Xinje XCPPro project, PLC1: XC3-60 (software 3.3k)

PROGRAM Ladder

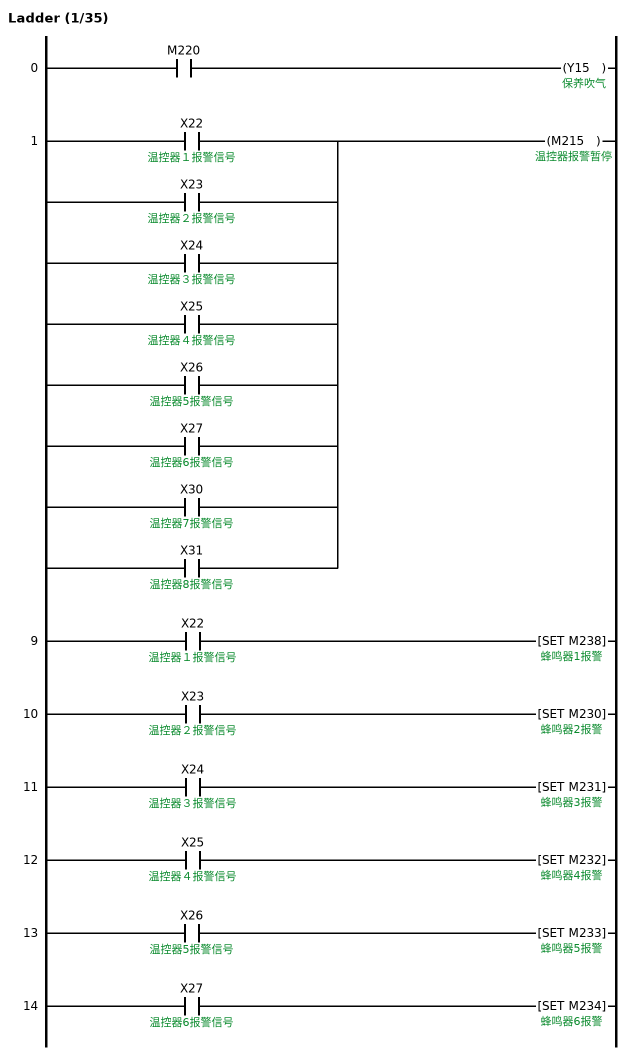
LD     M220
OUT    Y15	; 保养吹气 
LD     X22	; 温控器１报警信号
OR     X23	; 温控器２报警信号
OR     X24	; 温控器３报警信号
OR     X25	; 温控器４报警信号
OR     X26	; 温控器5报警信号
OR     X27	; 温控器6报警信号
OR     X30	; 温控器7报警信号
OR     X31	; 温控器8报警信号
OUT    M215	; 温控器报警暂停
LD     X22	; 温控器１报警信号
SET    M238	; 蜂鸣器1报警
LD     X23	; 温控器２报警信号
SET    M230	; 蜂鸣器2报警
LD     X24	; 温控器３报警信号
SET    M231	; 蜂鸣器3报警
LD     X25	; 温控器４报警信号
SET    M232	; 蜂鸣器4报警
LD     X26	; 温控器5报警信号
SET    M233	; 蜂鸣器5报警
LD     X27	; 温控器6报警信号
SET    M234	; 蜂鸣器6报警

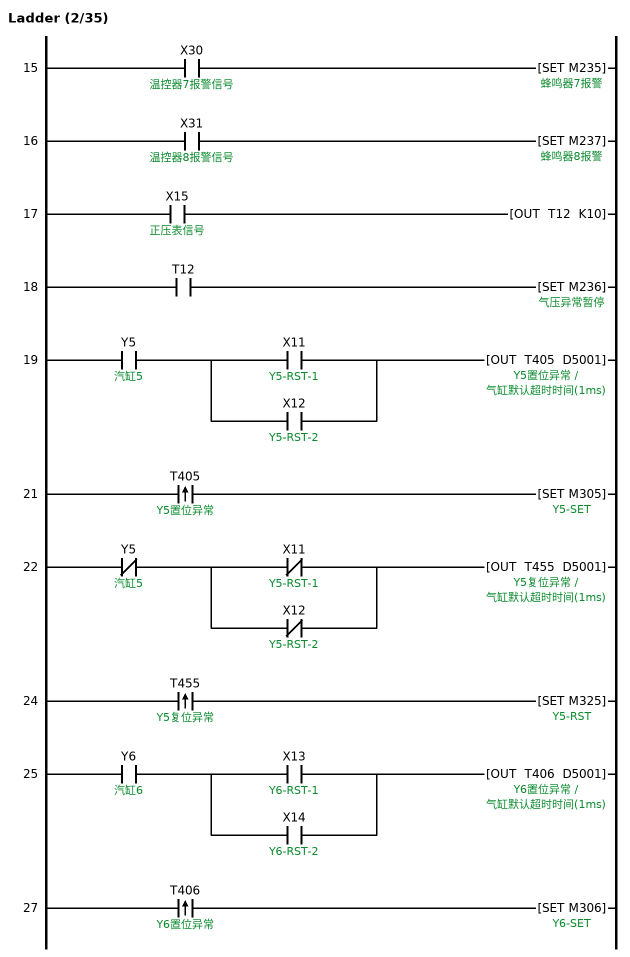
LD     X30	; 温控器7报警信号
SET    M235	; 蜂鸣器7报警
LD     X31	; 温控器8报警信号
SET    M237	; 蜂鸣器8报警
LD     X15	; 正压表信号
OUT    T12 K10
LD     T12
SET    M236	; 气压异常暂停
LD     Y5	; 汽缸5
LD     X11	; Y5-RST-1
OR     X12	; Y5-RST-2
ANB
OUT    T405 D5001	; Y5置位异常 / 气缸默认超时时间(1ms)
LDP    T405	; Y5置位异常
SET    M305	; Y5-SET
LDI    Y5	; 汽缸5
LDI    X11	; Y5-RST-1
ORI    X12	; Y5-RST-2
ANB
OUT    T455 D5001	; Y5复位异常 / 气缸默认超时时间(1ms)
LDP    T455	; Y5复位异常
SET    M325	; Y5-RST
LD     Y6	; 汽缸6
LD     X13	; Y6-RST-1
OR     X14	; Y6-RST-2
ANB
OUT    T406 D5001	; Y6置位异常 / 气缸默认超时时间(1ms)
LDP    T406	; Y6置位异常
SET    M306	; Y6-SET

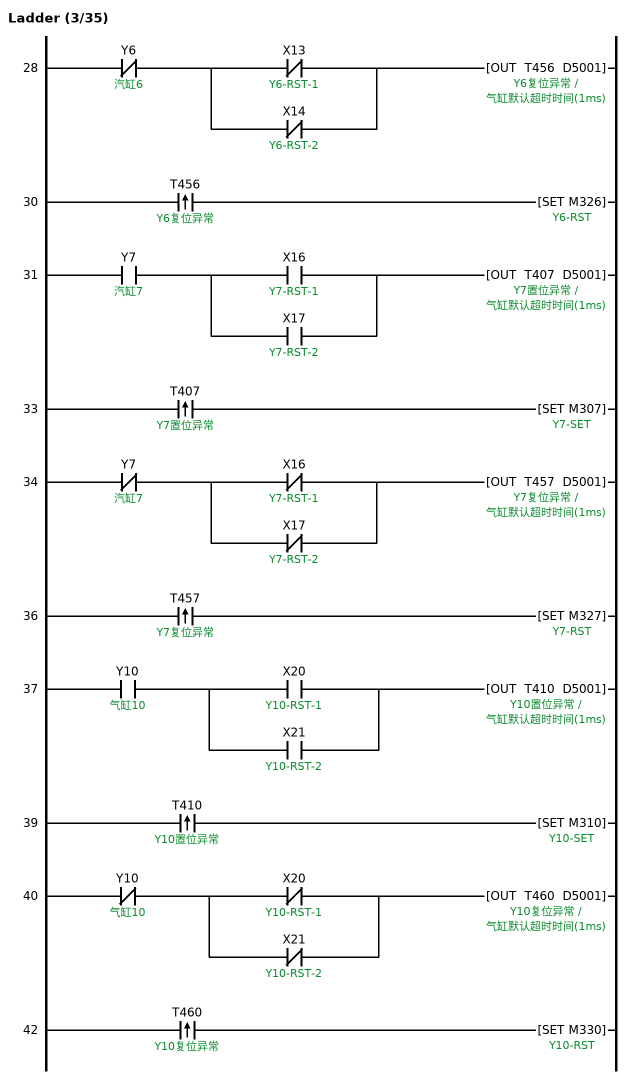
LDI    Y6	; 汽缸6
LDI    X13	; Y6-RST-1
ORI    X14	; Y6-RST-2
ANB
OUT    T456 D5001	; Y6复位异常 / 气缸默认超时时间(1ms)
LDP    T456	; Y6复位异常
SET    M326	; Y6-RST
LD     Y7	; 汽缸7
LD     X16	; Y7-RST-1
OR     X17	; Y7-RST-2
ANB
OUT    T407 D5001	; Y7置位异常 / 气缸默认超时时间(1ms)
LDP    T407	; Y7置位异常
SET    M307	; Y7-SET
LDI    Y7	; 汽缸7
LDI    X16	; Y7-RST-1
ORI    X17	; Y7-RST-2
ANB
OUT    T457 D5001	; Y7复位异常 / 气缸默认超时时间(1ms)
LDP    T457	; Y7复位异常
SET    M327	; Y7-RST
LD     Y10	; 气缸10
LD     X20	; Y10-RST-1
OR     X21	; Y10-RST-2
ANB
OUT    T410 D5001	; Y10置位异常 / 气缸默认超时时间(1ms)
LDP    T410	; Y10置位异常
SET    M310	; Y10-SET
LDI    Y10	; 气缸10
LDI    X20	; Y10-RST-1
ORI    X21	; Y10-RST-2
ANB
OUT    T460 D5001	; Y10复位异常 / 气缸默认超时时间(1ms)
LDP    T460	; Y10复位异常
SET    M330	; Y10-RST

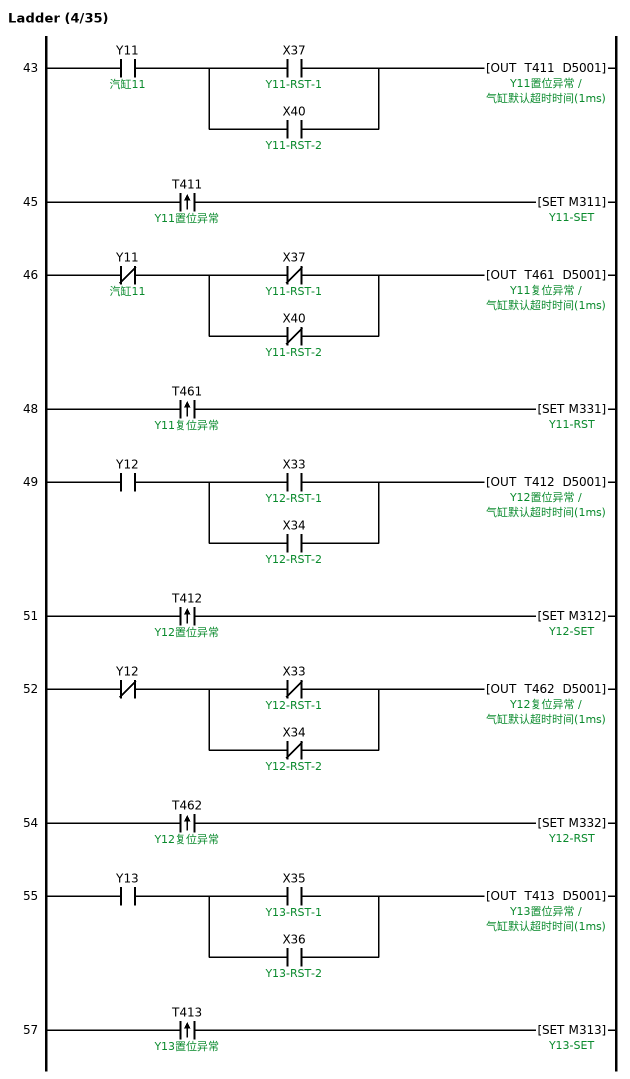
LD     Y11	; 汽缸11
LD     X37	; Y11-RST-1
OR     X40	; Y11-RST-2
ANB
OUT    T411 D5001	; Y11置位异常 / 气缸默认超时时间(1ms)
LDP    T411	; Y11置位异常
SET    M311	; Y11-SET
LDI    Y11	; 汽缸11
LDI    X37	; Y11-RST-1
ORI    X40	; Y11-RST-2
ANB
OUT    T461 D5001	; Y11复位异常 / 气缸默认超时时间(1ms)
LDP    T461	; Y11复位异常
SET    M331	; Y11-RST
LD     Y12
LD     X33	; Y12-RST-1
OR     X34	; Y12-RST-2
ANB
OUT    T412 D5001	; Y12置位异常 / 气缸默认超时时间(1ms)
LDP    T412	; Y12置位异常
SET    M312	; Y12-SET
LDI    Y12
LDI    X33	; Y12-RST-1
ORI    X34	; Y12-RST-2
ANB
OUT    T462 D5001	; Y12复位异常 / 气缸默认超时时间(1ms)
LDP    T462	; Y12复位异常
SET    M332	; Y12-RST
LD     Y13
LD     X35	; Y13-RST-1
OR     X36	; Y13-RST-2
ANB
OUT    T413 D5001	; Y13置位异常 / 气缸默认超时时间(1ms)
LDP    T413	; Y13置位异常
SET    M313	; Y13-SET

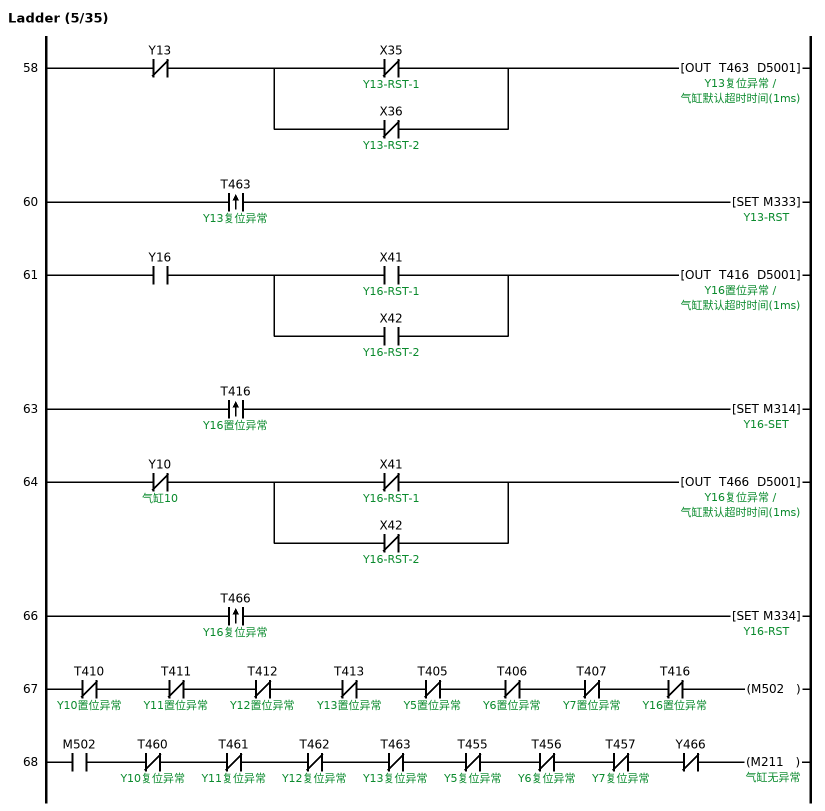
LDI    Y13
LDI    X35	; Y13-RST-1
ORI    X36	; Y13-RST-2
ANB
OUT    T463 D5001	; Y13复位异常 / 气缸默认超时时间(1ms)
LDP    T463	; Y13复位异常
SET    M333	; Y13-RST
LD     Y16
LD     X41	; Y16-RST-1
OR     X42	; Y16-RST-2
ANB
OUT    T416 D5001	; Y16置位异常 / 气缸默认超时时间(1ms)
LDP    T416	; Y16置位异常
SET    M314	; Y16-SET
LDI    Y10	; 气缸10
LDI    X41	; Y16-RST-1
ORI    X42	; Y16-RST-2
ANB
OUT    T466 D5001	; Y16复位异常 / 气缸默认超时时间(1ms)
LDP    T466	; Y16复位异常
SET    M334	; Y16-RST
LDI    T410	; Y10置位异常
ANI    T411	; Y11置位异常
ANI    T412	; Y12置位异常
ANI    T413	; Y13置位异常
ANI    T405	; Y5置位异常
ANI    T406	; Y6置位异常
ANI    T407	; Y7置位异常
ANI    T416	; Y16置位异常
OUT    M502
LD     M502
ANI    T460	; Y10复位异常
ANI    T461	; Y11复位异常
ANI    T462	; Y12复位异常
ANI    T463	; Y13复位异常
ANI    T455	; Y5复位异常
ANI    T456	; Y6复位异常
ANI    T457	; Y7复位异常
ANI    Y466
OUT    M211	; 气缸无异常

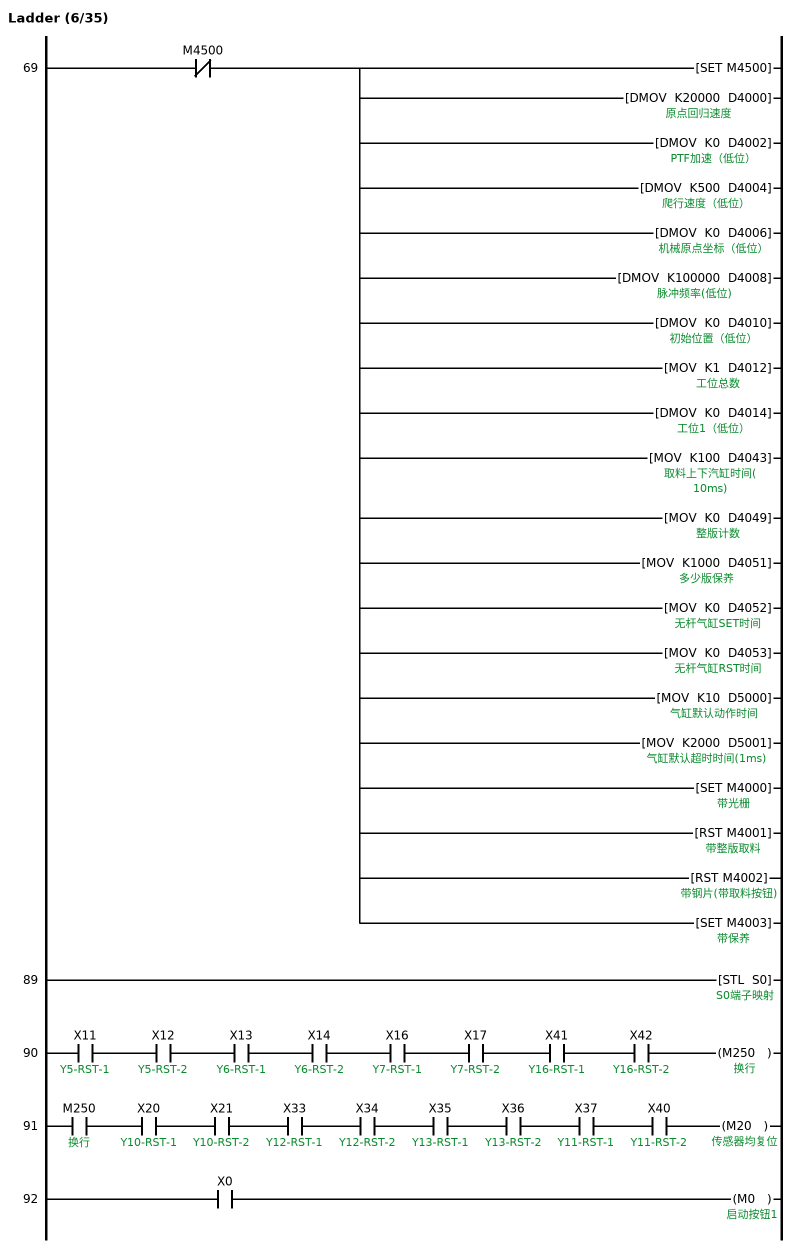
LDI    M4500
SET    M4500
DMOV   K20000 D4000	; 原点回归速度
DMOV   K0 D4002	; PTF加速（低位）
DMOV   K500 D4004	; 爬行速度（低位）
DMOV   K0 D4006	; 机械原点坐标（低位）
DMOV   K100000 D4008	; 脉冲频率(低位)
DMOV   K0 D4010	; 初始位置（低位）
MOV    K1 D4012	; 工位总数
DMOV   K0 D4014	; 工位1（低位）
MOV    K100 D4043	; 取料上下汽缸时间(10ms)
MOV    K0 D4049	; 整版计数
MOV    K1000 D4051	; 多少版保养
MOV    K0 D4052	; 无杆气缸SET时间
MOV    K0 D4053	; 无杆气缸RST时间
MOV    K10 D5000	; 气缸默认动作时间
MOV    K2000 D5001	; 气缸默认超时时间(1ms)
SET    M4000	; 带光栅
RST    M4001	; 带整版取料
RST    M4002	; 带钢片(带取料按钮)
SET    M4003	; 带保养
STL    S0	; S0端子映射
LD     X11	; Y5-RST-1
AND    X12	; Y5-RST-2
AND    X13	; Y6-RST-1
AND    X14	; Y6-RST-2
AND    X16	; Y7-RST-1
AND    X17	; Y7-RST-2
AND    X41	; Y16-RST-1
AND    X42	; Y16-RST-2
OUT    M250	; 换行
LD     M250	; 换行
AND    X20	; Y10-RST-1
AND    X21	; Y10-RST-2
AND    X33	; Y12-RST-1
AND    X34	; Y12-RST-2
AND    X35	; Y13-RST-1
AND    X36	; Y13-RST-2
AND    X37	; Y11-RST-1
AND    X40	; Y11-RST-2
OUT    M20	; 传感器均复位
LD     X0
OUT    M0	; 启动按钮1

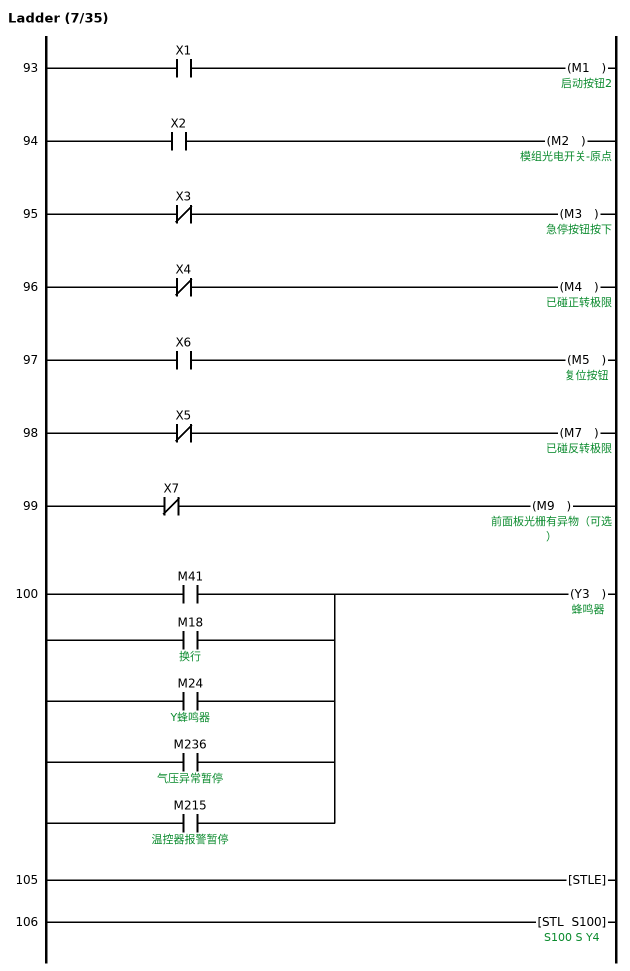
LD     X1
OUT    M1	; 启动按钮2
LD     X2
OUT    M2	; 模组光电开关-原点
LDI    X3
OUT    M3	; 急停按钮按下
LDI    X4
OUT    M4	; 已碰正转极限
LD     X6
OUT    M5	; 复位按钮
LDI    X5
OUT    M7	; 已碰反转极限
LDI    X7
OUT    M9	; 前面板光栅有异物（可选）
LD     M41
OR     M18	; 换行
OR     M24	; Y蜂鸣器
OR     M236	; 气压异常暂停
OR     M215	; 温控器报警暂停
OUT    Y3	; 蜂鸣器
STLE
STL    S100	; S100 S Y4

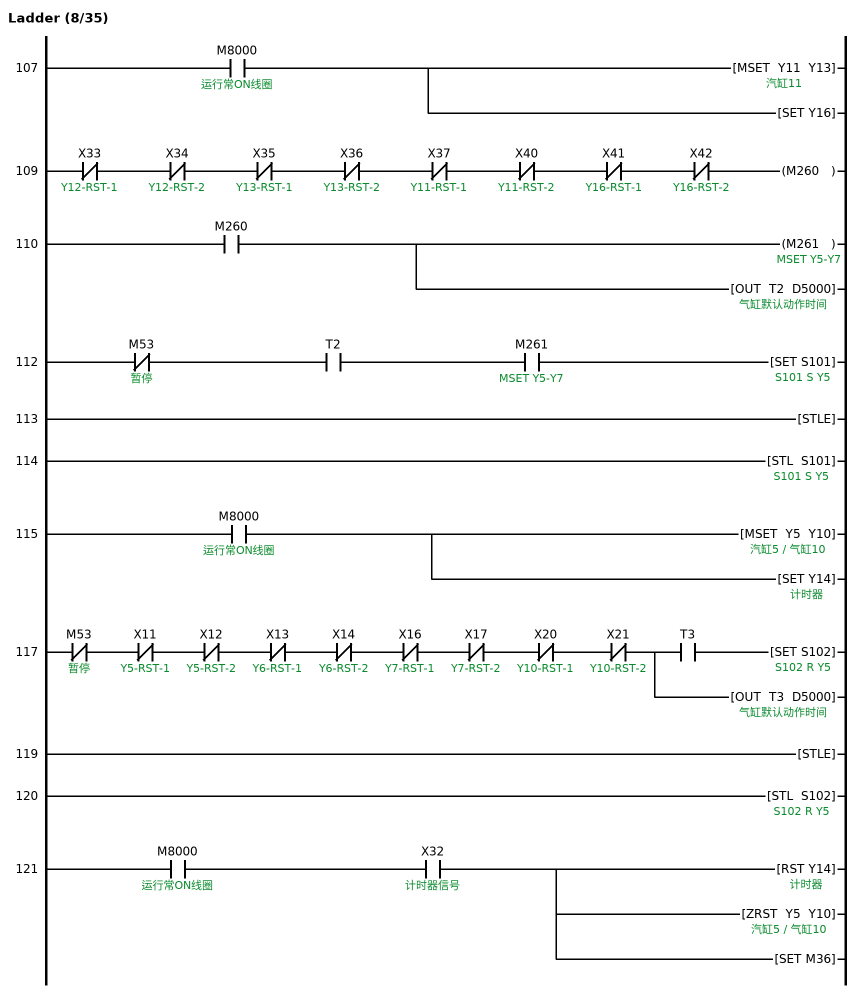
LD     M8000	; 运行常ON线圈
MSET   Y11 Y13	; 汽缸11
SET    Y16
LDI    X33	; Y12-RST-1
ANI    X34	; Y12-RST-2
ANI    X35	; Y13-RST-1
ANI    X36	; Y13-RST-2
ANI    X37	; Y11-RST-1
ANI    X40	; Y11-RST-2
ANI    X41	; Y16-RST-1
ANI    X42	; Y16-RST-2
OUT    M260
LD     M260
OUT    M261	; MSET Y5-Y7
OUT    T2 D5000	; 气缸默认动作时间
LDI    M53	; 暂停
AND    T2
AND    M261	; MSET Y5-Y7
SET    S101	; S101 S Y5
STLE
STL    S101	; S101 S Y5
LD     M8000	; 运行常ON线圈
MSET   Y5 Y10	; 汽缸5 / 气缸10
SET    Y14	; 计时器
LDI    M53	; 暂停
ANI    X11	; Y5-RST-1
ANI    X12	; Y5-RST-2
ANI    X13	; Y6-RST-1
ANI    X14	; Y6-RST-2
ANI    X16	; Y7-RST-1
ANI    X17	; Y7-RST-2
ANI    X20	; Y10-RST-1
ANI    X21	; Y10-RST-2
MPS
AND    T3
SET    S102	; S102 R Y5 
MPP
OUT    T3 D5000	; 气缸默认动作时间
STLE
STL    S102	; S102 R Y5 
LD     M8000	; 运行常ON线圈
AND    X32	; 计时器信号
RST    Y14	; 计时器
ZRST   Y5 Y10	; 汽缸5 / 气缸10
SET    M36

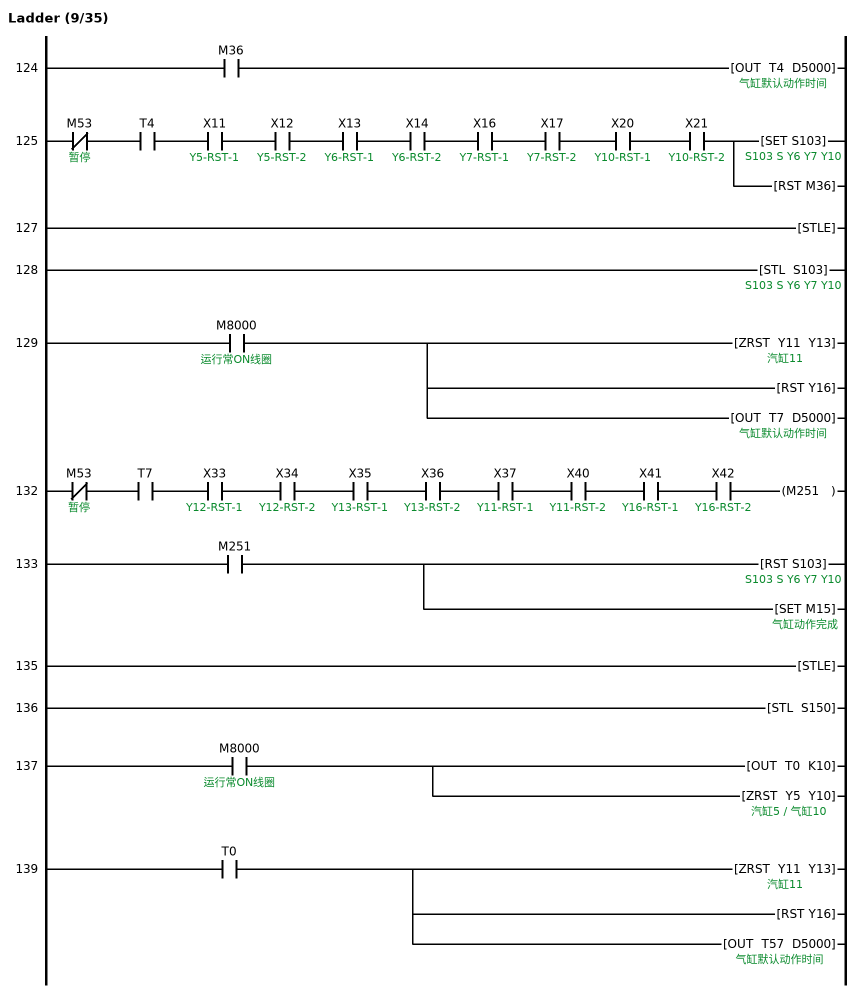
LD     M36
OUT    T4 D5000	; 气缸默认动作时间
LDI    M53	; 暂停
AND    T4
AND    X11	; Y5-RST-1
AND    X12	; Y5-RST-2
AND    X13	; Y6-RST-1
AND    X14	; Y6-RST-2
AND    X16	; Y7-RST-1
AND    X17	; Y7-RST-2
AND    X20	; Y10-RST-1
AND    X21	; Y10-RST-2
SET    S103	; S103 S Y6 Y7 Y10 
RST    M36
STLE
STL    S103	; S103 S Y6 Y7 Y10 
LD     M8000	; 运行常ON线圈
ZRST   Y11 Y13	; 汽缸11
RST    Y16
OUT    T7 D5000	; 气缸默认动作时间
LDI    M53	; 暂停
AND    T7
AND    X33	; Y12-RST-1
AND    X34	; Y12-RST-2
AND    X35	; Y13-RST-1
AND    X36	; Y13-RST-2
AND    X37	; Y11-RST-1
AND    X40	; Y11-RST-2
AND    X41	; Y16-RST-1
AND    X42	; Y16-RST-2
OUT    M251
LD     M251
RST    S103	; S103 S Y6 Y7 Y10 
SET    M15	; 气缸动作完成
STLE
STL    S150
LD     M8000	; 运行常ON线圈
OUT    T0 K10
ZRST   Y5 Y10	; 汽缸5 / 气缸10
LD     T0
ZRST   Y11 Y13	; 汽缸11
RST    Y16
OUT    T57 D5000	; 气缸默认动作时间

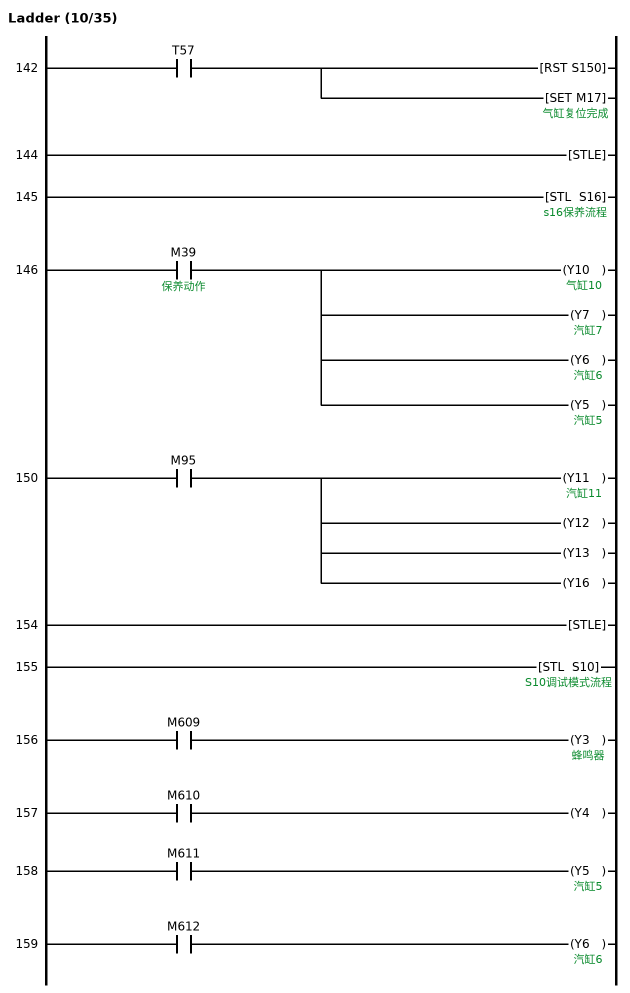
LD     T57
RST    S150
SET    M17	; 气缸复位完成
STLE
STL    S16	; s16保养流程
LD     M39	; 保养动作
OUT    Y10	; 气缸10
OUT    Y7	; 汽缸7
OUT    Y6	; 汽缸6
OUT    Y5	; 汽缸5
LD     M95
OUT    Y11	; 汽缸11
OUT    Y12
OUT    Y13
OUT    Y16
STLE
STL    S10	; S10调试模式流程
LD     M609
OUT    Y3	; 蜂鸣器
LD     M610
OUT    Y4
LD     M611
OUT    Y5	; 汽缸5
LD     M612
OUT    Y6	; 汽缸6

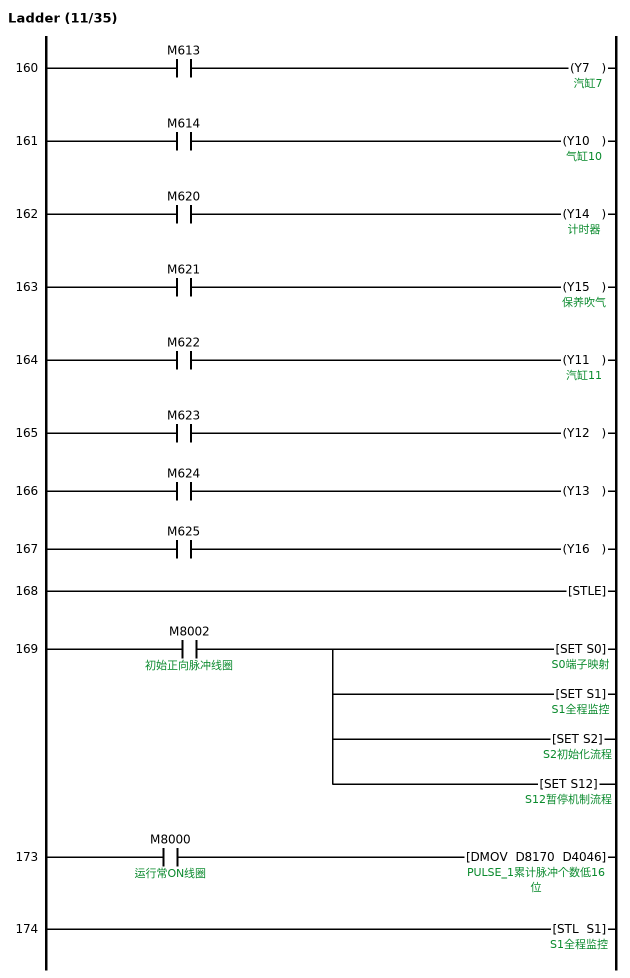
LD     M613
OUT    Y7	; 汽缸7
LD     M614
OUT    Y10	; 气缸10
LD     M620
OUT    Y14	; 计时器
LD     M621
OUT    Y15	; 保养吹气 
LD     M622
OUT    Y11	; 汽缸11
LD     M623
OUT    Y12
LD     M624
OUT    Y13
LD     M625
OUT    Y16
STLE
LD     M8002	; 初始正向脉冲线圈
SET    S0	; S0端子映射
SET    S1	; S1全程监控
SET    S2	; S2初始化流程
SET    S12	; S12暂停机制流程
LD     M8000	; 运行常ON线圈
DMOV   D8170 D4046	; PULSE_1累计脉冲个数低16位
STL    S1	; S1全程监控

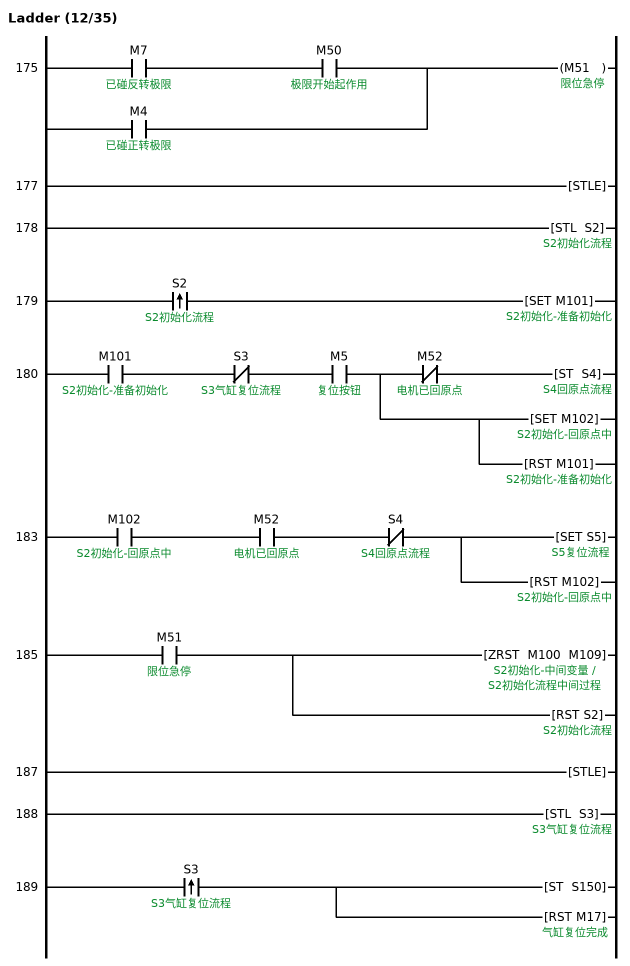
LD     M7	; 已碰反转极限
AND    M50	; 极限开始起作用
OR     M4	; 已碰正转极限
OUT    M51	; 限位急停
STLE
STL    S2	; S2初始化流程
LDP    S2	; S2初始化流程
SET    M101	; S2初始化-准备初始化
LD     M101	; S2初始化-准备初始化
ANI    S3	; S3气缸复位流程
AND    M5	; 复位按钮
MPS
ANI    M52	; 电机已回原点
ST     S4	; S4回原点流程
MPP
SET    M102	; S2初始化-回原点中
RST    M101	; S2初始化-准备初始化
LD     M102	; S2初始化-回原点中
AND    M52	; 电机已回原点
ANI    S4	; S4回原点流程
SET    S5	; S5复位流程
RST    M102	; S2初始化-回原点中
LD     M51	; 限位急停
ZRST   M100 M109	; S2初始化-中间变量 / S2初始化流程中间过程
RST    S2	; S2初始化流程
STLE
STL    S3	; S3气缸复位流程
LDP    S3	; S3气缸复位流程
ST     S150
RST    M17	; 气缸复位完成

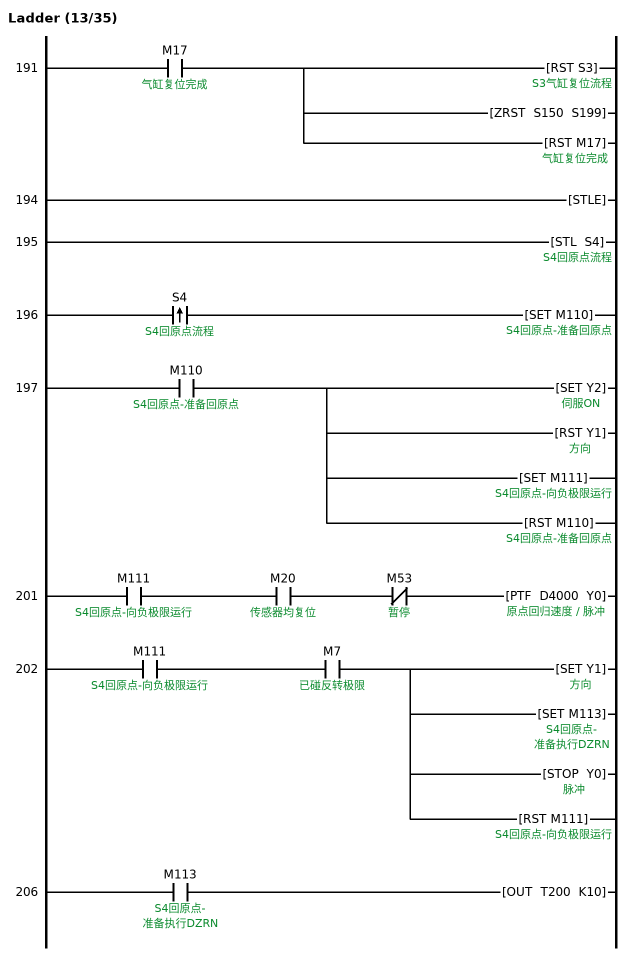
LD     M17	; 气缸复位完成
RST    S3	; S3气缸复位流程
ZRST   S150 S199
RST    M17	; 气缸复位完成
STLE
STL    S4	; S4回原点流程
LDP    S4	; S4回原点流程
SET    M110	; S4回原点-准备回原点
LD     M110	; S4回原点-准备回原点
SET    Y2	; 伺服ON
RST    Y1	; 方向
SET    M111	; S4回原点-向负极限运行
RST    M110	; S4回原点-准备回原点
LD     M111	; S4回原点-向负极限运行
AND    M20	; 传感器均复位
ANI    M53	; 暂停
PTF    D4000 Y0	; 原点回归速度 / 脉冲
LD     M111	; S4回原点-向负极限运行
AND    M7	; 已碰反转极限
SET    Y1	; 方向
SET    M113	; S4回原点-准备执行DZRN
STOP   Y0	; 脉冲
RST    M111	; S4回原点-向负极限运行
LD     M113	; S4回原点-准备执行DZRN
OUT    T200 K10

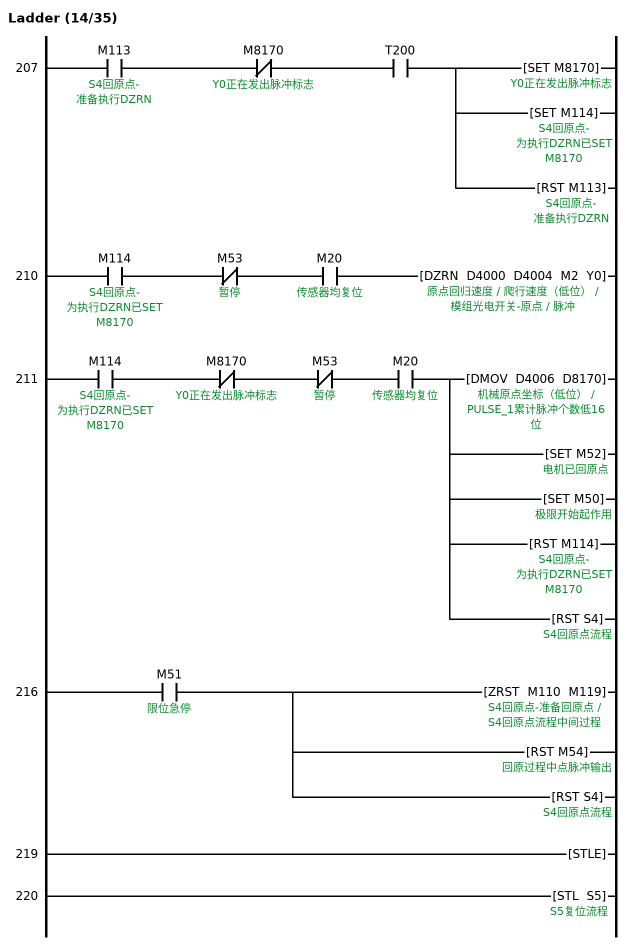
LD     M113	; S4回原点-准备执行DZRN
ANI    M8170	; Y0正在发出脉冲标志
AND    T200
SET    M8170	; Y0正在发出脉冲标志
SET    M114	; S4回原点-为执行DZRN已SET M8170
RST    M113	; S4回原点-准备执行DZRN
LD     M114	; S4回原点-为执行DZRN已SET M8170
ANI    M53	; 暂停
AND    M20	; 传感器均复位
DZRN   D4000 D4004 M2 Y0	; 原点回归速度 / 爬行速度（低位） / 模组光电开关-原点 / 脉冲
LD     M114	; S4回原点-为执行DZRN已SET M8170
ANI    M8170	; Y0正在发出脉冲标志
ANI    M53	; 暂停
AND    M20	; 传感器均复位
DMOV   D4006 D8170	; 机械原点坐标（低位） / PULSE_1累计脉冲个数低16位
SET    M52	; 电机已回原点
SET    M50	; 极限开始起作用
RST    M114	; S4回原点-为执行DZRN已SET M8170
RST    S4	; S4回原点流程
LD     M51	; 限位急停
ZRST   M110 M119	; S4回原点-准备回原点 / S4回原点流程中间过程
RST    M54	; 回原过程中点脉冲输出
RST    S4	; S4回原点流程
STLE
STL    S5	; S5复位流程

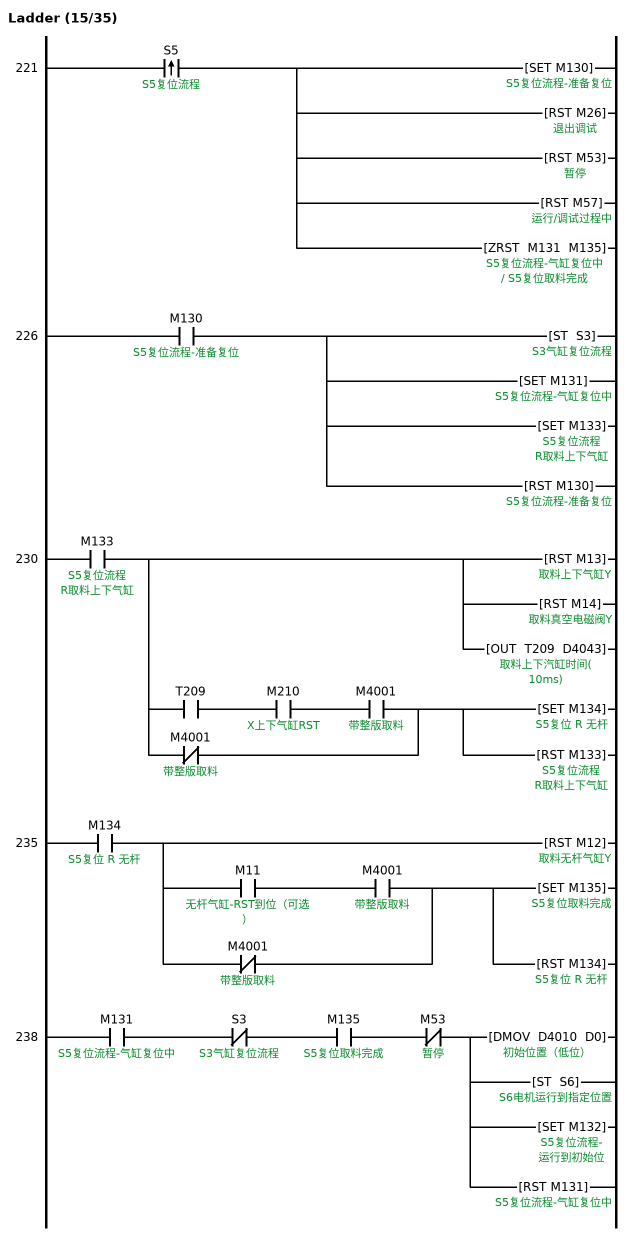
LDP    S5	; S5复位流程
SET    M130	; S5复位流程-准备复位
RST    M26	; 退出调试
RST    M53	; 暂停
RST    M57	; 运行/调试过程中
ZRST   M131 M135	; S5复位流程-气缸复位中 / S5复位取料完成
LD     M130	; S5复位流程-准备复位
ST     S3	; S3气缸复位流程
SET    M131	; S5复位流程-气缸复位中
SET    M133	; S5复位流程 R取料上下气缸
RST    M130	; S5复位流程-准备复位
LD     M133	; S5复位流程 R取料上下气缸
RST    M13	; 取料上下气缸Y
RST    M14	; 取料真空电磁阀Y
OUT    T209 D4043	; 取料上下汽缸时间(10ms)
LD     T209
AND    M210	; X上下气缸RST
AND    M4001	; 带整版取料
ORI    M4001	; 带整版取料
ANB
SET    M134	; S5复位 R 无杆
RST    M133	; S5复位流程 R取料上下气缸
LD     M134	; S5复位 R 无杆
RST    M12	; 取料无杆气缸Y
LD     M11	; 无杆气缸-RST到位（可选）
AND    M4001	; 带整版取料
ORI    M4001	; 带整版取料
ANB
SET    M135	; S5复位取料完成
RST    M134	; S5复位 R 无杆
LD     M131	; S5复位流程-气缸复位中
ANI    S3	; S3气缸复位流程
AND    M135	; S5复位取料完成
ANI    M53	; 暂停
DMOV   D4010 D0	; 初始位置（低位）
ST     S6	; S6电机运行到指定位置
SET    M132	; S5复位流程-运行到初始位
RST    M131	; S5复位流程-气缸复位中

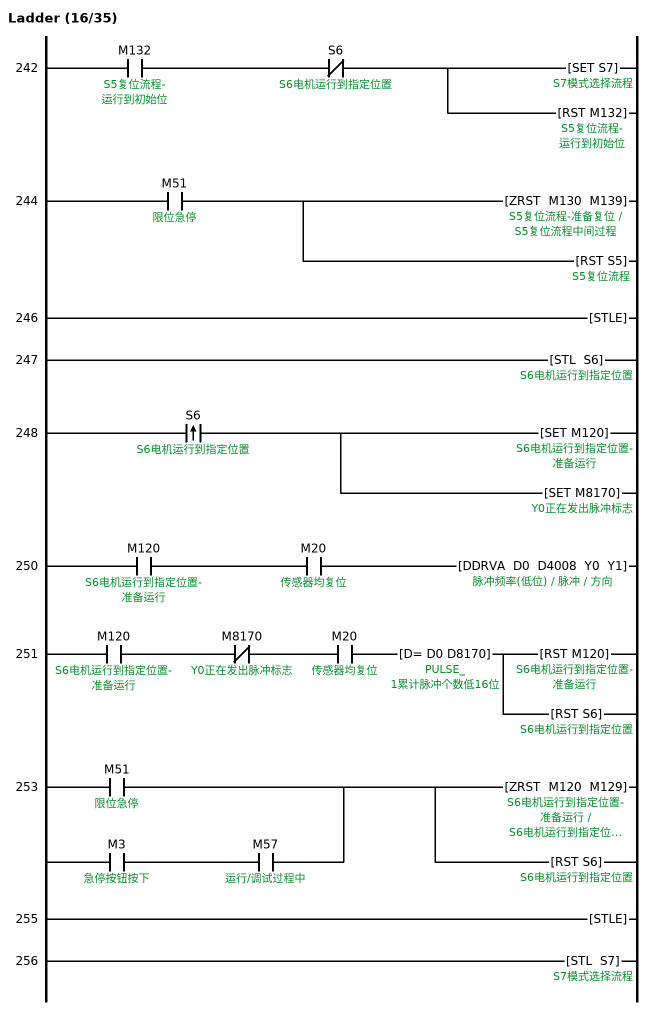
LD     M132	; S5复位流程-运行到初始位
ANI    S6	; S6电机运行到指定位置
SET    S7	; S7模式选择流程
RST    M132	; S5复位流程-运行到初始位
LD     M51	; 限位急停
ZRST   M130 M139	; S5复位流程-准备复位 / S5复位流程中间过程
RST    S5	; S5复位流程
STLE
STL    S6	; S6电机运行到指定位置
LDP    S6	; S6电机运行到指定位置
SET    M120	; S6电机运行到指定位置-准备运行
SET    M8170	; Y0正在发出脉冲标志
LD     M120	; S6电机运行到指定位置-准备运行
AND    M20	; 传感器均复位
DDRVA  D0 D4008 Y0 Y1	; 脉冲频率(低位) / 脉冲 / 方向
LD     M120	; S6电机运行到指定位置-准备运行
ANI    M8170	; Y0正在发出脉冲标志
AND    M20	; 传感器均复位
DAND=  D0 D8170	; PULSE_1累计脉冲个数低16位
RST    M120	; S6电机运行到指定位置-准备运行
RST    S6	; S6电机运行到指定位置
LD     M51	; 限位急停
LD     M3	; 急停按钮按下
AND    M57	; 运行/调试过程中
ORB
ZRST   M120 M129	; S6电机运行到指定位置-准备运行 / S6电机运行到指定位置中间过程
RST    S6	; S6电机运行到指定位置
STLE
STL    S7	; S7模式选择流程

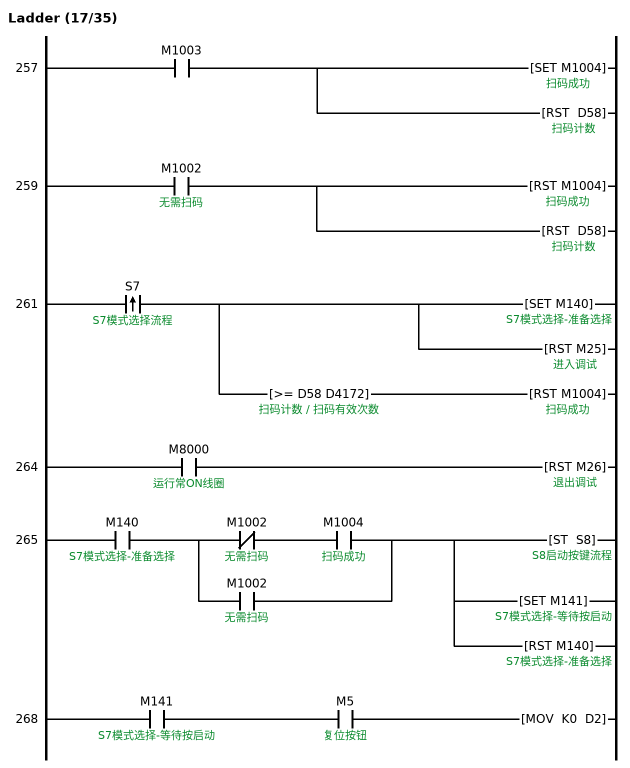
LD     M1003
SET    M1004	; 扫码成功
RST    D58	; 扫码计数
LD     M1002	; 无需扫码
RST    M1004	; 扫码成功
RST    D58	; 扫码计数
LDP    S7	; S7模式选择流程
SET    M140	; S7模式选择-准备选择
RST    M25	; 进入调试
AND>=  D58 D4172	; 扫码计数 / 扫码有效次数
RST    M1004	; 扫码成功
LD     M8000	; 运行常ON线圈
RST    M26	; 退出调试
LD     M140	; S7模式选择-准备选择
LDI    M1002	; 无需扫码
AND    M1004	; 扫码成功
OR     M1002	; 无需扫码
ANB
ST     S8	; S8启动按键流程
SET    M141	; S7模式选择-等待按启动
RST    M140	; S7模式选择-准备选择
LD     M141	; S7模式选择-等待按启动
AND    M5	; 复位按钮
MOV    K0 D2

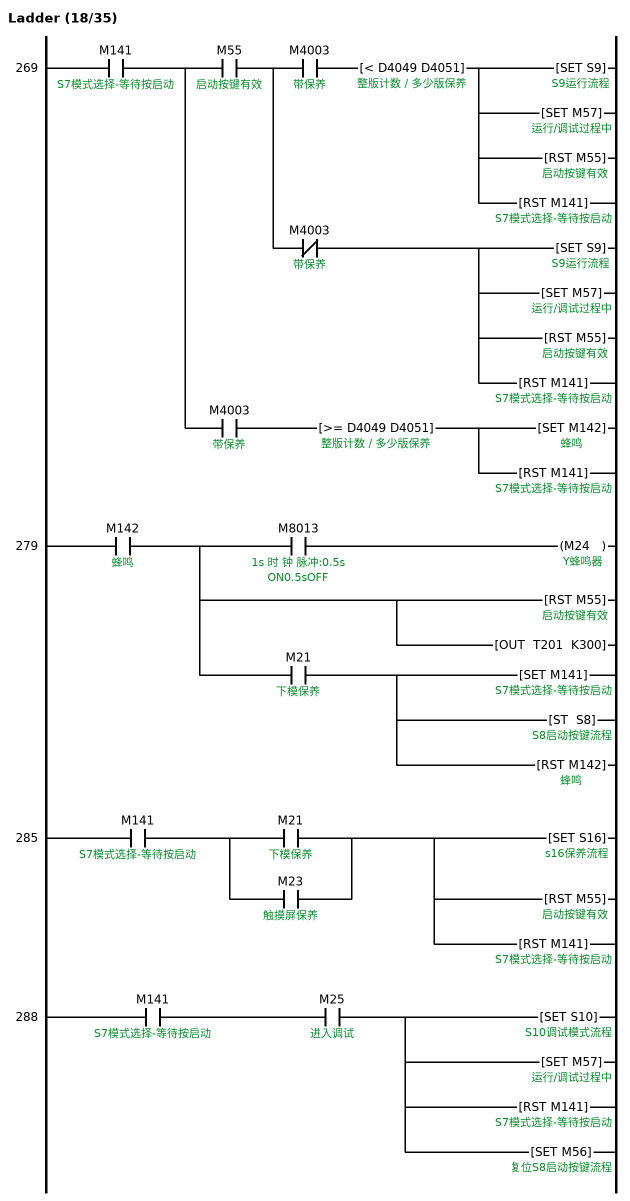
LD     M141	; S7模式选择-等待按启动
MPS
AND    M55	; 启动按键有效
MPS
AND    M4003	; 带保养
AND<   D4049 D4051	; 整版计数 / 多少版保养
SET    S9	; S9运行流程
SET    M57	; 运行/调试过程中
RST    M55	; 启动按键有效
RST    M141	; S7模式选择-等待按启动
MPP
ANI    M4003	; 带保养
SET    S9	; S9运行流程
SET    M57	; 运行/调试过程中
RST    M55	; 启动按键有效
RST    M141	; S7模式选择-等待按启动
MPP
AND    M4003	; 带保养
AND>=  D4049 D4051	; 整版计数 / 多少版保养
SET    M142	; 蜂鸣
RST    M141	; S7模式选择-等待按启动
LD     M142	; 蜂鸣
MPS
AND    M8013	; 1s 时 钟 脉冲:0.5s ON0.5sOFF
OUT    M24	; Y蜂鸣器
MPP
RST    M55	; 启动按键有效
OUT    T201 K300
AND    M21	; 下模保养
SET    M141	; S7模式选择-等待按启动
ST     S8	; S8启动按键流程
RST    M142	; 蜂鸣
LD     M141	; S7模式选择-等待按启动
LD     M21	; 下模保养
OR     M23	; 触摸屏保养
ANB
SET    S16	; s16保养流程
RST    M55	; 启动按键有效
RST    M141	; S7模式选择-等待按启动
LD     M141	; S7模式选择-等待按启动
AND    M25	; 进入调试
SET    S10	; S10调试模式流程
SET    M57	; 运行/调试过程中
RST    M141	; S7模式选择-等待按启动
SET    M56	; 复位S8启动按键流程

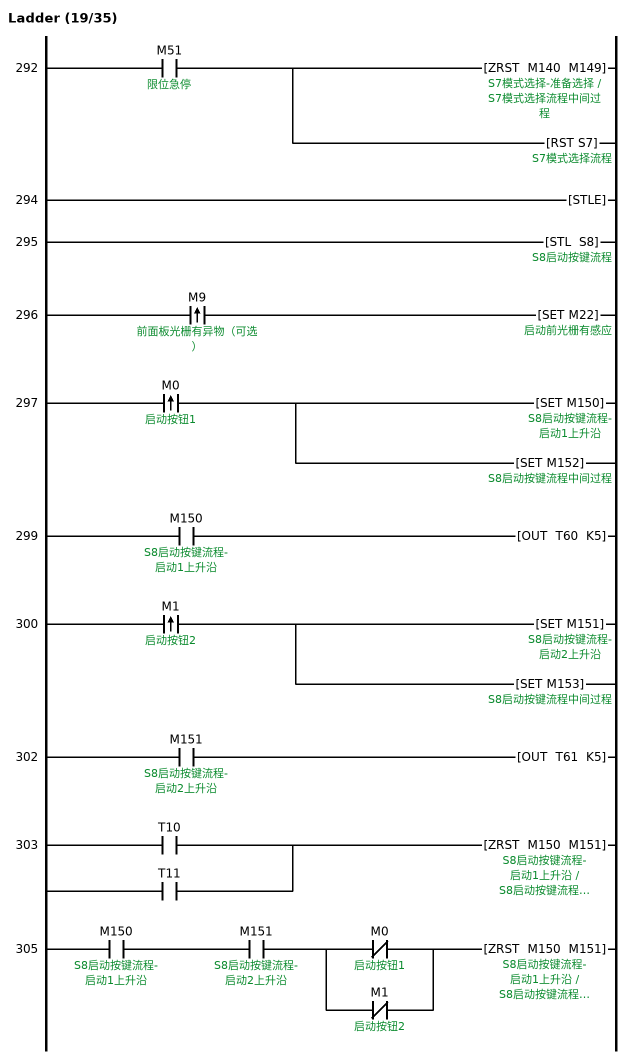
LD     M51	; 限位急停
ZRST   M140 M149	; S7模式选择-准备选择 / S7模式选择流程中间过程
RST    S7	; S7模式选择流程
STLE
STL    S8	; S8启动按键流程
LDP    M9	; 前面板光栅有异物（可选）
SET    M22	; 启动前光栅有感应
LDP    M0	; 启动按钮1
SET    M150	; S8启动按键流程-启动1上升沿
SET    M152	; S8启动按键流程中间过程
LD     M150	; S8启动按键流程-启动1上升沿
OUT    T60 K5
LDP    M1	; 启动按钮2
SET    M151	; S8启动按键流程-启动2上升沿
SET    M153	; S8启动按键流程中间过程
LD     M151	; S8启动按键流程-启动2上升沿
OUT    T61 K5
LD     T10
OR     T11
ZRST   M150 M151	; S8启动按键流程-启动1上升沿 / S8启动按键流程-启动2上升沿
LD     M150	; S8启动按键流程-启动1上升沿
AND    M151	; S8启动按键流程-启动2上升沿
LDI    M0	; 启动按钮1
ORI    M1	; 启动按钮2
ANB
ZRST   M150 M151	; S8启动按键流程-启动1上升沿 / S8启动按键流程-启动2上升沿

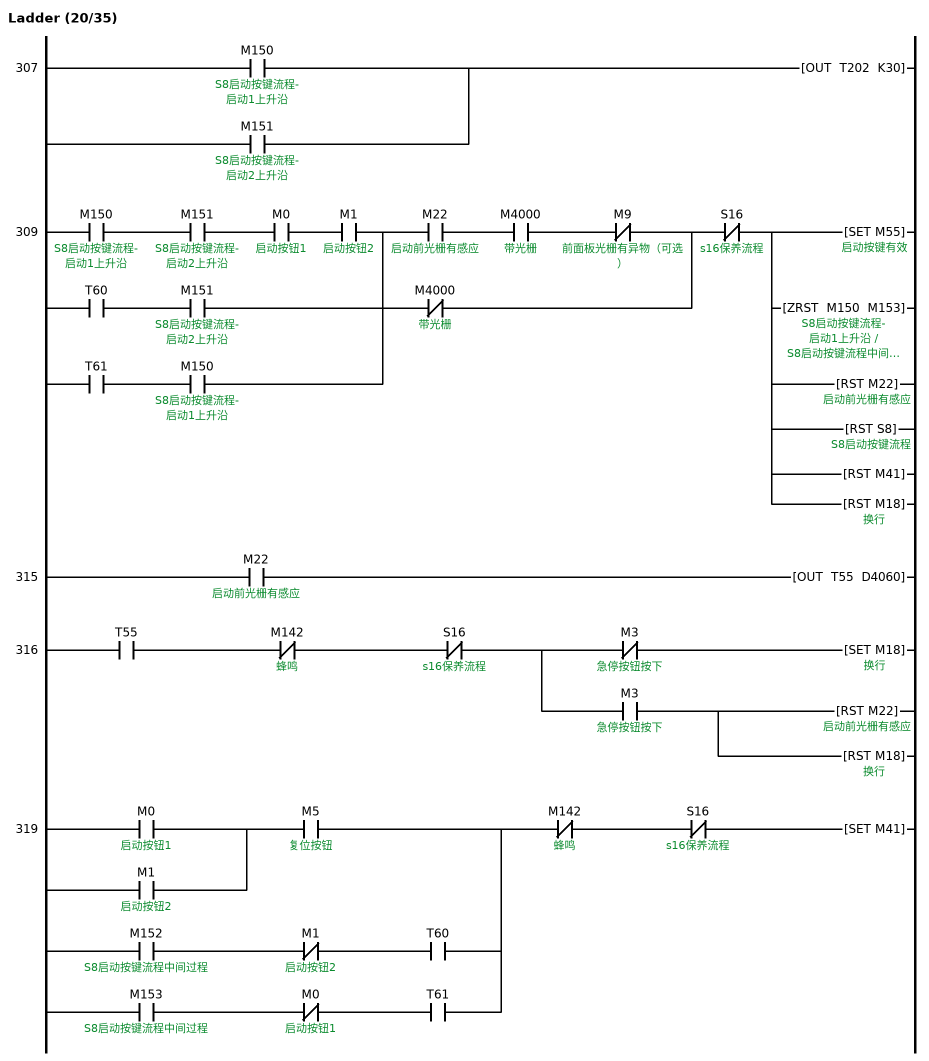
LD     M150	; S8启动按键流程-启动1上升沿
OR     M151	; S8启动按键流程-启动2上升沿
OUT    T202 K30
LD     M150	; S8启动按键流程-启动1上升沿
AND    M151	; S8启动按键流程-启动2上升沿
AND    M0	; 启动按钮1
AND    M1	; 启动按钮2
LD     T60
AND    M151	; S8启动按键流程-启动2上升沿
ORB
LD     T61
AND    M150	; S8启动按键流程-启动1上升沿
ORB
LD     M22	; 启动前光栅有感应
AND    M4000	; 带光栅
ANI    M9	; 前面板光栅有异物（可选）
ORI    M4000	; 带光栅
ANB
ANI    S16	; s16保养流程
SET    M55	; 启动按键有效
ZRST   M150 M153	; S8启动按键流程-启动1上升沿 / S8启动按键流程中间过程
RST    M22	; 启动前光栅有感应
RST    S8	; S8启动按键流程
RST    M41
RST    M18	; 换行
LD     M22	; 启动前光栅有感应
OUT    T55 D4060
LD     T55
ANI    M142	; 蜂鸣
ANI    S16	; s16保养流程
MPS
ANI    M3	; 急停按钮按下
SET    M18	; 换行
MPP
AND    M3	; 急停按钮按下
RST    M22	; 启动前光栅有感应
RST    M18	; 换行
LD     M0	; 启动按钮1
OR     M1	; 启动按钮2
AND    M5	; 复位按钮
LD     M152	; S8启动按键流程中间过程
ANI    M1	; 启动按钮2
AND    T60
ORB
LD     M153	; S8启动按键流程中间过程
ANI    M0	; 启动按钮1
AND    T61
ORB
ANI    M142	; 蜂鸣
ANI    S16	; s16保养流程
SET    M41

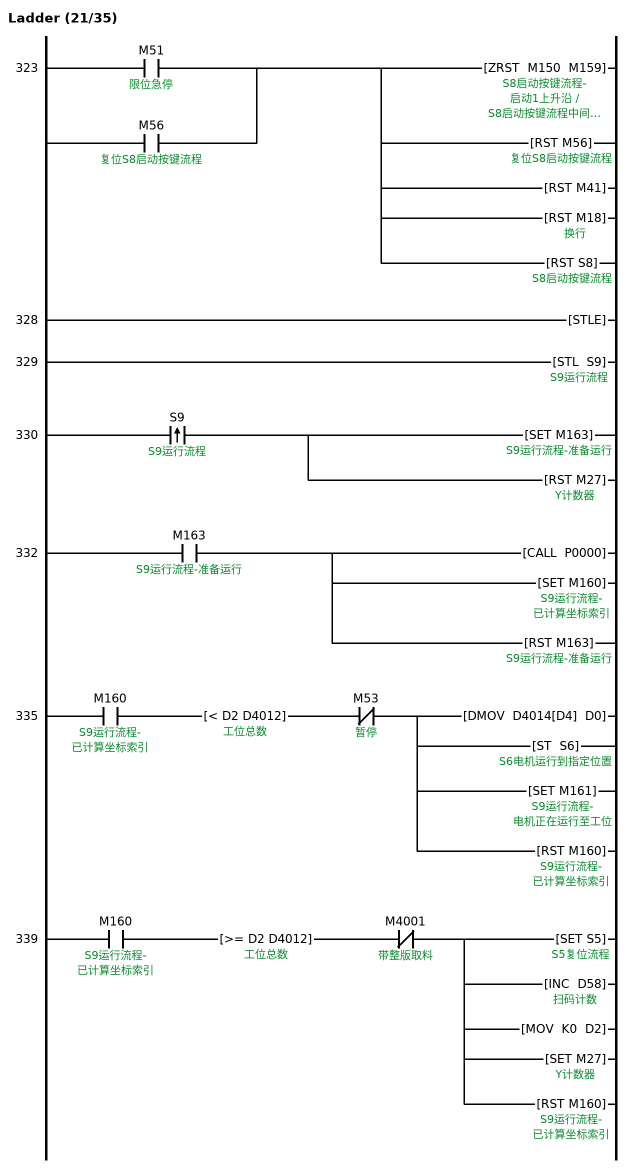
LD     M51	; 限位急停
OR     M56	; 复位S8启动按键流程
ZRST   M150 M159	; S8启动按键流程-启动1上升沿 / S8启动按键流程中间过程
RST    M56	; 复位S8启动按键流程
RST    M41
RST    M18	; 换行
RST    S8	; S8启动按键流程
STLE
STL    S9	; S9运行流程
LDP    S9	; S9运行流程
SET    M163	; S9运行流程-准备运行
RST    M27	; Y计数器
LD     M163	; S9运行流程-准备运行
CALL   P0000
SET    M160	; S9运行流程-已计算坐标索引
RST    M163	; S9运行流程-准备运行
LD     M160	; S9运行流程-已计算坐标索引
AND<   D2 D4012	; 工位总数
ANI    M53	; 暂停
DMOV   D4014[D4] D0
ST     S6	; S6电机运行到指定位置
SET    M161	; S9运行流程-电机正在运行至工位
RST    M160	; S9运行流程-已计算坐标索引
LD     M160	; S9运行流程-已计算坐标索引
AND>=  D2 D4012	; 工位总数
ANI    M4001	; 带整版取料
SET    S5	; S5复位流程
INC    D58	; 扫码计数
MOV    K0 D2
SET    M27	; Y计数器
RST    M160	; S9运行流程-已计算坐标索引

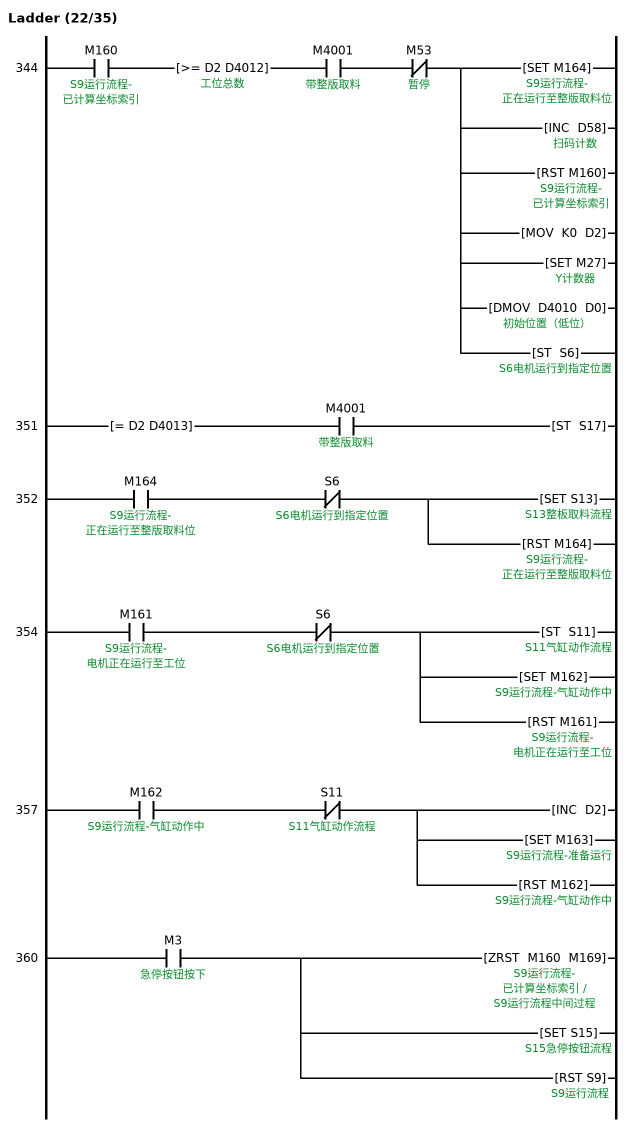
LD     M160	; S9运行流程-已计算坐标索引
AND>=  D2 D4012	; 工位总数
AND    M4001	; 带整版取料
ANI    M53	; 暂停
SET    M164	; S9运行流程-正在运行至整版取料位
INC    D58	; 扫码计数
RST    M160	; S9运行流程-已计算坐标索引
MOV    K0 D2
SET    M27	; Y计数器
DMOV   D4010 D0	; 初始位置（低位）
ST     S6	; S6电机运行到指定位置
LD=    D2 D4013
AND    M4001	; 带整版取料
ST     S17
LD     M164	; S9运行流程-正在运行至整版取料位
ANI    S6	; S6电机运行到指定位置
SET    S13	; S13整板取料流程
RST    M164	; S9运行流程-正在运行至整版取料位
LD     M161	; S9运行流程-电机正在运行至工位
ANI    S6	; S6电机运行到指定位置
ST     S11	; S11气缸动作流程
SET    M162	; S9运行流程-气缸动作中
RST    M161	; S9运行流程-电机正在运行至工位
LD     M162	; S9运行流程-气缸动作中
ANI    S11	; S11气缸动作流程
INC    D2
SET    M163	; S9运行流程-准备运行
RST    M162	; S9运行流程-气缸动作中
LD     M3	; 急停按钮按下
ZRST   M160 M169	; S9运行流程-已计算坐标索引 / S9运行流程中间过程
SET    S15	; S15急停按钮流程
RST    S9	; S9运行流程

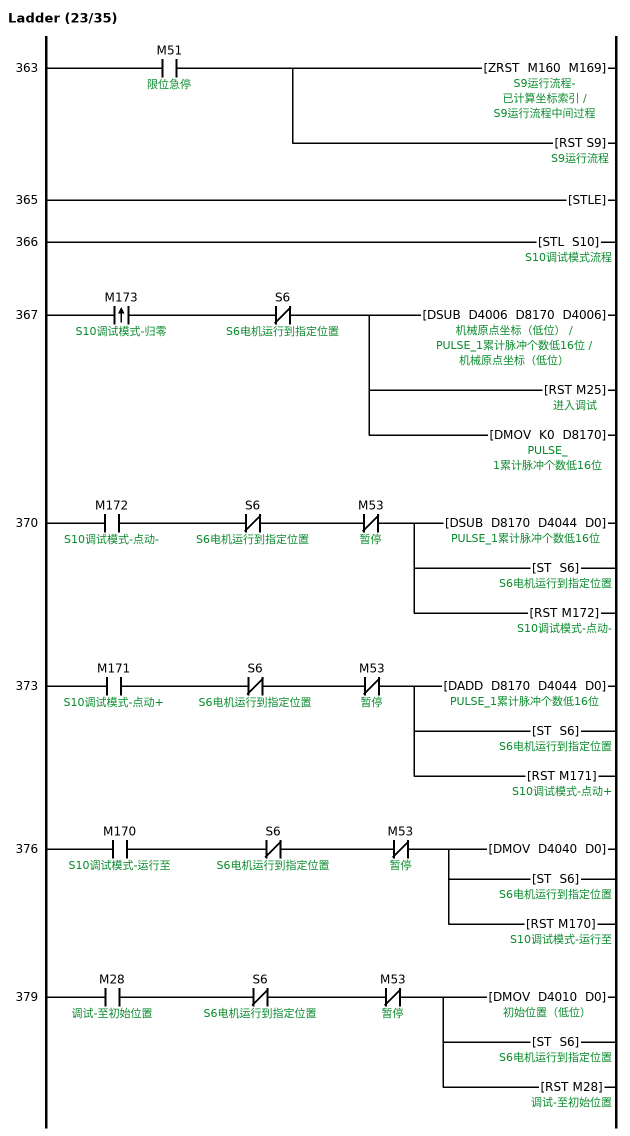
LD     M51	; 限位急停
ZRST   M160 M169	; S9运行流程-已计算坐标索引 / S9运行流程中间过程
RST    S9	; S9运行流程
STLE
STL    S10	; S10调试模式流程
LDP    M173	; S10调试模式-归零
ANI    S6	; S6电机运行到指定位置
DSUB   D4006 D8170 D4006	; 机械原点坐标（低位） / PULSE_1累计脉冲个数低16位 / 机械原点坐标（低位）
RST    M25	; 进入调试
DMOV   K0 D8170	; PULSE_1累计脉冲个数低16位
LD     M172	; S10调试模式-点动-
ANI    S6	; S6电机运行到指定位置
ANI    M53	; 暂停
DSUB   D8170 D4044 D0	; PULSE_1累计脉冲个数低16位
ST     S6	; S6电机运行到指定位置
RST    M172	; S10调试模式-点动-
LD     M171	; S10调试模式-点动+
ANI    S6	; S6电机运行到指定位置
ANI    M53	; 暂停
DADD   D8170 D4044 D0	; PULSE_1累计脉冲个数低16位
ST     S6	; S6电机运行到指定位置
RST    M171	; S10调试模式-点动+
LD     M170	; S10调试模式-运行至
ANI    S6	; S6电机运行到指定位置
ANI    M53	; 暂停
DMOV   D4040 D0
ST     S6	; S6电机运行到指定位置
RST    M170	; S10调试模式-运行至
LD     M28	; 调试-至初始位置
ANI    S6	; S6电机运行到指定位置
ANI    M53	; 暂停
DMOV   D4010 D0	; 初始位置（低位）
ST     S6	; S6电机运行到指定位置
RST    M28	; 调试-至初始位置

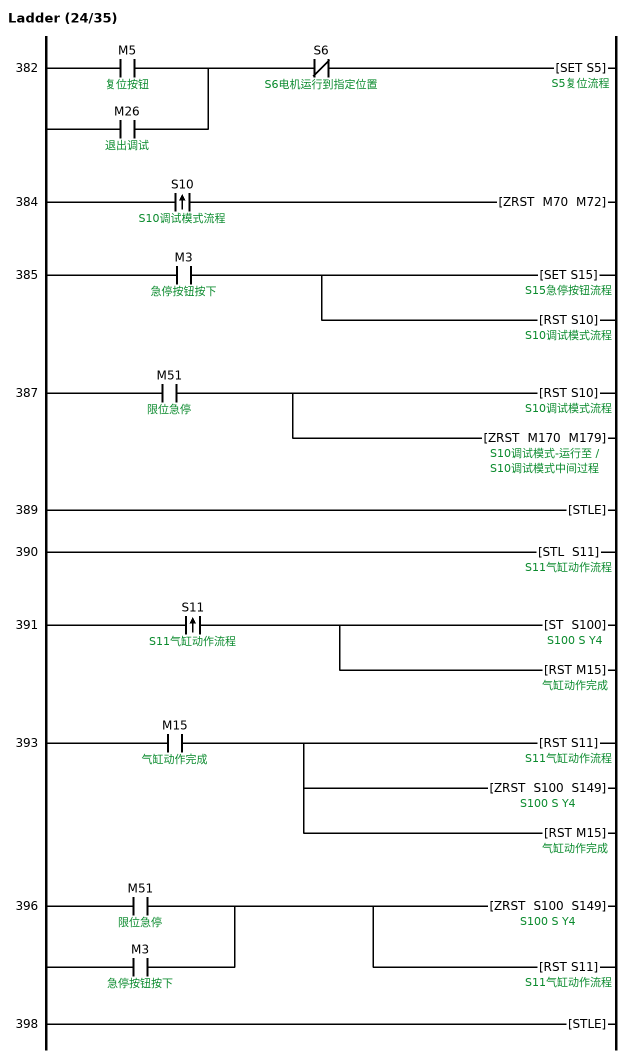
LD     M5	; 复位按钮
OR     M26	; 退出调试
ANI    S6	; S6电机运行到指定位置
SET    S5	; S5复位流程
LDP    S10	; S10调试模式流程
ZRST   M70 M72
LD     M3	; 急停按钮按下
SET    S15	; S15急停按钮流程
RST    S10	; S10调试模式流程
LD     M51	; 限位急停
RST    S10	; S10调试模式流程
ZRST   M170 M179	; S10调试模式-运行至 / S10调试模式中间过程
STLE
STL    S11	; S11气缸动作流程
LDP    S11	; S11气缸动作流程
ST     S100	; S100 S Y4
RST    M15	; 气缸动作完成
LD     M15	; 气缸动作完成
RST    S11	; S11气缸动作流程
ZRST   S100 S149	; S100 S Y4
RST    M15	; 气缸动作完成
LD     M51	; 限位急停
OR     M3	; 急停按钮按下
ZRST   S100 S149	; S100 S Y4
RST    S11	; S11气缸动作流程
STLE

